(* IEC 61131-3 sources: simple-control-modules/test, 8 files *)

(* ---- AbstractEncoderTest.st ---- *)
USING AxUnit.Assert;
USING Simatic.Ax.SimpleControlModules;

NAMESPACE Simatic.Ax.SimpleControlModules
    CLASS EncoderTest EXTENDS Simatic.Ax.SimpleControlModules.AbstractEncoder
        VAR

        END_VAR

        METHOD PUBLIC OVERRIDE Evaluate
            ;
        END_METHOD
    END_CLASS
END_NAMESPACE

NAMESPACE Simatic.Ax.SimpleControlModules.Test
    {TestFixture}
    CLASS Test_AbstractEncoder

        VAR
            enc : EncoderTest;
        END_VAR

        {Test}
        METHOD PUBLIC SetValue_to_555_expect_GetValue_555

            enc.SetValue(LINT#555);

            Equal(expected := LINT#555, actual := enc.GetValue());
            Equal(expected := LINT#0, actual := enc.RelativeCount());
            enc.Reset();

            Equal(expected := LINT#0, actual := enc.GetValue());
            Equal(expected := LINT#0, actual := enc.RelativeCount());
        END_METHOD

        {Test}
        METHOD PUBLIC Test_Reset_Expect_value_0

            enc.SetValue(LINT#555);
            enc.Reset();

            Equal(expected := LINT#0, actual := enc.GetValue());
            Equal(expected := LINT#0, actual := enc.RelativeCount());
        END_METHOD

    END_CLASS

END_NAMESPACE

(* ---- CounterTest.st ---- *)
USING AxUnit.Assert;
USING AxUnit.Assert;
USING Simatic.Ax.SimpleControlModules;
NAMESPACE Simatic.Ax.SimpleControlModules.Test
    {TestFixture}
    CLASS TestCounterClass
        VAR
            cnt : Counter;
            cntStateLess : Counter;
        END_VAR

        {TestSetup}
        METHOD PUBLIC MyTestSetup
            // Will be called before MyTest_A AND before Test_B are executed
            cnt := cntStateLess;
        END_METHOD

        {Test}
        METHOD PUBLIC Count_Forward_3_times_Expect_3;
            cnt.CountForward();
            Equal(expected := 1, actual := cnt.CounterValue());
            cnt.CountForward();
            cnt.CountForward();
            Equal(expected := 3, actual := cnt.CounterValue());
        END_METHOD

        {Test}
        METHOD PUBLIC Count_Reverse_3_times_From_3_Expect_0;
            cnt.SetCounterValue(value := 3);
            Equal(expected := 3, actual := cnt.CounterValue());
            cnt.CountReverse();
            Equal(expected := 2, actual := cnt.CounterValue());
            cnt.CountReverse();
            cnt.CountReverse();
            Equal(expected := 0, actual := cnt.CounterValue());
        END_METHOD

        {Test}
        METHOD PUBLIC Count_Forward_3_times_by_2_Expect_3;
            cnt.CountForward(increment := 2);
            Equal(expected := 2, actual := cnt.CounterValue());
            cnt.CountForward(increment := 2);
            cnt.CountForward(increment := 2);
            Equal(expected := 6, actual := cnt.CounterValue());
        END_METHOD

        {Test}
        METHOD PUBLIC Count_Reverse_3_timesby_2_From_6_Expect_0;
            cnt.SetCounterValue(value := 6);
            Equal(expected := 6, actual := cnt.CounterValue());
            cnt.CountReverse(decrement := 2);
            Equal(expected := 4, actual := cnt.CounterValue());
            cnt.CountReverse(decrement := 2);
            cnt.CountReverse(decrement := 2);
            Equal(expected := 0, actual := cnt.CounterValue());
        END_METHOD

        {Test}
        METHOD PUBLIC Counter_Lower_Limit_Reached
            cnt.Config(ll := DINT#-4, ul := DINT#4);
            Equal(expected := FALSE, actual := cnt.LowerLimitReached());
            Equal(expected := FALSE, actual := cnt.UpperLimitReached());
            cnt.CountReverse();
            cnt.CountReverse();
            cnt.CountReverse();
            Equal(expected := FALSE, actual := cnt.LowerLimitReached());
            cnt.CountReverse();
            Equal(expected := TRUE, actual := cnt.LowerLimitReached());
            Equal(expected := FALSE, actual := cnt.UpperLimitReached());
        END_METHOD

        {Test}
        METHOD PUBLIC Counter_Lower_Limit_Reached_When_Limit_Is_1
            cnt.Config(ll := DINT#1, ul := DINT#4);
            Equal(expected := TRUE, actual := cnt.LowerLimitReached());
            Equal(expected := FALSE, actual := cnt.UpperLimitReached());
            cnt.CountReverse();
            cnt.CountReverse();
            cnt.CountReverse();
            Equal(expected := TRUE, actual := cnt.LowerLimitReached());
            cnt.CountReverse();
            Equal(expected := TRUE, actual := cnt.LowerLimitReached());
            Equal(expected := FALSE, actual := cnt.UpperLimitReached());
        END_METHOD

        {Test}
        METHOD PUBLIC Counter_Upper_Limit_Reached_When_UpperLimit_Is4
            cnt.Config(ll := DINT#-4, ul := DINT#4);
            Equal(expected := FALSE, actual := cnt.LowerLimitReached());
            Equal(expected := FALSE, actual := cnt.UpperLimitReached());
            cnt.CountForward();
            cnt.CountForward();
            cnt.CountForward();
            Equal(expected := FALSE, actual := cnt.UpperLimitReached());
            cnt.CountForward();
            Equal(expected := TRUE, actual := cnt.UpperLimitReached());
            Equal(expected := FALSE, actual := cnt.LowerLimitReached());
            cnt.CountReverse();
            Equal(expected := FALSE, actual := cnt.UpperLimitReached());
        END_METHOD

        {Test}
        METHOD PUBLIC Counter_Upper_Limit_Reached_When_UpperLimit_Is0
            cnt.Config(ll := DINT#-4, ul := DINT#0);
            Equal(expected := FALSE, actual := cnt.LowerLimitReached());
            Equal(expected := TRUE, actual := cnt.UpperLimitReached());
            cnt.CountForward();
            cnt.CountForward();
            cnt.CountForward();
            Equal(expected := TRUE, actual := cnt.UpperLimitReached());
            cnt.CountForward();
            Equal(expected := TRUE, actual := cnt.UpperLimitReached());
            Equal(expected := FALSE, actual := cnt.LowerLimitReached());
        END_METHOD
    END_CLASS
END_NAMESPACE

(* ---- EncoderABTest.st ---- *)
USING Simatic.Ax.IO.Input;
USING AxUnit.Assert;
USING Simatic.Ax.SimpleControlModules;
NAMESPACE Simatic.Ax.SimpleControlModules.Test
    {TestFixture}
    CLASS Test_EncoderAB IMPLEMENTS AxUnit.Mocking.IPayload

        VAR
            enc : EncoderAB;
            sigA : BinSignal;
            sigB : BinSignal;
            //signalMock : BinSignalQMockAB;

            signalsA : ARRAY[0..13] OF BOOL := [FALSE, TRUE, TRUE, FALSE, FALSE, TRUE, TRUE, FALSE, FALSE, TRUE, TRUE, FALSE, FALSE, TRUE];
            signalsB : ARRAY[0..13] OF BOOL := [FALSE, FALSE, TRUE, TRUE, FALSE, FALSE, TRUE, TRUE, FALSE, FALSE, TRUE, TRUE, FALSE, FALSE];

        END_VAR

        {Test}
        // Encoder Forward Test
        METHOD PUBLIC AB_Encoder_A_Forward_test_Expect_13
                VAR_TEMP
                    i : INT;
                END_VAR

                enc.SignalA := sigA;
                enc.SignalB := sigB;

                FOR i := 0 TO 13 DO
                    sigA.ReadCyclic(signal := signalsA[i]);
                    sigB.ReadCyclic(signal := signalsB[i]);
                    enc.Evaluate();
                END_FOR;

                Equal(expected := LINT#13, actual := enc.GetValue());
                Equal(expected := LINT#13, actual := enc.RelativeCount());
                ;
        END_METHOD

        // Encoder Count Reverse Test
        {Test}
        METHOD PUBLIC AB_Encoder_A_Reverse_test_Expect_Minus_13
            VAR_TEMP
                i : INT;
            END_VAR

            enc.SignalA := sigA;
            enc.SignalB := sigB;
            enc.SetDirection(mode := CountMode#Reverse);
            FOR i := 0 TO 13 DO
                sigA.ReadCyclic(signal := signalsA[i]);
                sigB.ReadCyclic(signal := signalsB[i]);

                enc.Evaluate();
            END_FOR;

            Equal(expected := LINT#-13, actual := enc.GetValue());
            Equal(expected := LINT#-13, actual := enc.RelativeCount());
            ;
        END_METHOD

        {Test}
        // Encoder Swap singnals Test
        METHOD PUBLIC AB_Encoder_Swap_AB_Signal_And_Expect_Minus_13
                VAR_TEMP
                    i : INT;
                END_VAR

                // Swap AB
                enc.SignalA := sigB;
                enc.SignalB := sigA;
                FOR i := 0 TO 13 DO
                    sigA.ReadCyclic(signal := signalsA[i]);
                    sigB.ReadCyclic(signal := signalsB[i]);
                    enc.Evaluate();
                END_FOR;

                Equal(expected := LINT#-13, actual := enc.GetValue());
                Equal(expected := LINT#-13, actual := enc.RelativeCount());
                ;
        END_METHOD

        // Encoder change signal sequence to reverse
        {Test}
        METHOD PUBLIC AB_Encoder_9_Forward_5_Reverse_expect
            VAR_TEMP
                i : INT;
            END_VAR

            enc.SignalA := sigA;
            enc.SignalB := sigB;

            FOR i := 0 TO 9 DO
                sigA.ReadCyclic(signal := signalsA[i]);
                sigB.ReadCyclic(signal := signalsB[i]);
                enc.Evaluate();
            END_FOR;

            Equal(expected := LINT#9, actual := enc.GetValue());

            FOR i := 9 TO 0 BY -1 DO
                sigA.ReadCyclic(signal := signalsA[i]);
                sigB.ReadCyclic(signal := signalsB[i]);
                enc.Evaluate();
            END_FOR;
            Equal(expected := LINT#0, actual := enc.GetValue());
            Equal(expected := LINT#0, actual := enc.RelativeCount());
            ;
        END_METHOD

        // Encoder Reverse Test
        {Test}
        METHOD PUBLIC AB_Encoder_9_Forward_4_Reverse_expet_5
            VAR_TEMP
                i : INT;
            END_VAR

            enc.SignalA := sigA;
            enc.SignalB := sigB;

            FOR i := 0 TO 9 DO
                sigA.ReadCyclic(signal := signalsA[i]);
                sigB.ReadCyclic(signal := signalsB[i]);

                enc.Evaluate();
            END_FOR;
            Equal(expected := LINT#9, actual := enc.GetValue());

            enc.SetDirection(mode := CountMode#Reverse);
            FOR i := 10 TO 13 DO
                sigA.ReadCyclic(signal := signalsA[i]);
                sigB.ReadCyclic(signal := signalsB[i]);
            enc.Evaluate();
            END_FOR;
            Equal(expected := LINT#5, actual := enc.GetValue());
            Equal(expected := LINT#5, actual := enc.RelativeCount());
            ;
        END_METHOD

        {Test}
        METHOD PUBLIC Single_Track_Test_Reset
            VAR_TEMP
                i : INT;
            END_VAR

            THIS.AB_Encoder_A_Forward_test_Expect_13();

            enc.Reset();
            Equal(expected := LINT#0, actual := enc.GetValue());
        END_METHOD

        {Test}
        METHOD PUBLIC AB_Encoder_RelativeValue
            VAR_TEMP
                i : INT;
            END_VAR

            // 3 Rising edges 3 Falling edges --> 6 pulses
            enc.SignalA := sigA;
            enc.SignalB := sigB;

            FOR i := 0 TO 9 DO
                sigA.ReadCyclic(signal := signalsA[i]);
                sigB.ReadCyclic(signal := signalsB[i]);
            enc.Evaluate();
            END_FOR;
            Equal(expected := LINT#9, actual := enc.GetValue());
            Equal(expected := LINT#9, actual := enc.RelativeCount());
            enc.ResetRelative();

            FOR i := 10 TO 13 DO
                sigA.ReadCyclic(signal := signalsA[i]);
                sigB.ReadCyclic(signal := signalsB[i]);
            enc.Evaluate();
            END_FOR;
            Equal(expected := LINT#13, actual := enc.GetValue());
            Equal(expected := LINT#4, actual := enc.RelativeCount());
            ;
        END_METHOD

    END_CLASS

END_NAMESPACE

(* ---- EncoderATest.st ---- *)
USING Simatic.Ax.IO.Input;
USING AxUnit.Assert;
USING Simatic.Ax.SimpleControlModules;

NAMESPACE Simatic.Ax.SimpleControlModules.Test
    {TestFixture}
    CLASS Test_EncoderA IMPLEMENTS AxUnit.Mocking.IPayload

        VAR
            enc : EncoderA;
            sig : BinSignal;
            signalMock : BinSignalQMock;
        END_VAR

        {Test}
        // Encoder Forward Test
        METHOD PUBLIC Single_Track_Encoder_A_Forward_test_Expect_6
                VAR_TEMP
                    i : INT;
                END_VAR

                // 3 Rising edges 3 Falling edges --> 6 pulses
                enc.SignalA := sig;
                FOR i := 0 TO 13 DO
                    sig.ReadCyclic(signal := signalMock.Q());
                    enc.Evaluate();
                END_FOR;

                Equal(expected := LINT#6, actual := enc.GetValue());
                Equal(expected := LINT#6, actual := enc.RelativeCount());
                ;
        END_METHOD

        // Encoder Reverse Test
        {Test}
        METHOD PUBLIC Single_Track_Encoder_A_Reverse_test_Expect_Minus_6
            VAR_TEMP
                i : INT;
            END_VAR

            // 3 Rising edges 3 Falling edges --> 6 pulses
            enc.SignalA := sig;
            enc.SetDirection(mode := CountMode#Reverse);
            FOR i := 0 TO 13 DO
                sig.ReadCyclic(signal := signalMock.Q());
                enc.Evaluate();
            END_FOR;

            Equal(expected := LINT#-6, actual := enc.GetValue());
            Equal(expected := LINT#-6, actual := enc.RelativeCount());
            ;
        END_METHOD

        // Encoder Reverse Test
        {Test}
        METHOD PUBLIC Single_Track_Encoder_4_Forward_2_Reverse_expet_2
            VAR_TEMP
                i : INT;
            END_VAR

            // 3 Rising edges 3 Falling edges --> 6 pulses
            enc.SignalA := sig;
            FOR i := 0 TO 9 DO
                sig.ReadCyclic(signal := signalMock.Q());
                enc.Evaluate();
            END_FOR;
            Equal(expected := LINT#4, actual := enc.GetValue());

            enc.SetDirection(mode := CountMode#Reverse);
            FOR i := 0 TO 3 DO
                sig.ReadCyclic(signal := signalMock.Q());
                enc.Evaluate();
            END_FOR;
            Equal(expected := LINT#2, actual := enc.GetValue());
            Equal(expected := LINT#2, actual := enc.RelativeCount());
            ;
        END_METHOD

        {Test}
        METHOD PUBLIC Single_Track_Test_Reset
            VAR_TEMP
                i : INT;
            END_VAR

            THIS.Single_Track_Encoder_A_Forward_test_Expect_6();

            enc.Reset();
            Equal(expected := LINT#0, actual := enc.GetValue());
        END_METHOD

        {Test}
        METHOD PUBLIC Single_Track_Encoder_RelativeValue
            VAR_TEMP
                i : INT;
            END_VAR

            // 3 Rising edges 3 Falling edges --> 6 pulses
            enc.SignalA := sig;
            FOR i := 0 TO 9 DO
                sig.ReadCyclic(signal := signalMock.Q());
                enc.Evaluate();
            END_FOR;
            Equal(expected := LINT#4, actual := enc.GetValue());
            Equal(expected := LINT#4, actual := enc.RelativeCount());
            enc.ResetRelative();

            FOR i := 0 TO 3 DO
                sig.ReadCyclic(signal := signalMock.Q());
                enc.Evaluate();
            END_FOR;
            Equal(expected := LINT#6, actual := enc.GetValue());
            Equal(expected := LINT#2, actual := enc.RelativeCount());
            ;
        END_METHOD

    END_CLASS

    CLASS BinSignalQMock
        VAR PUBLIC
            signal : BOOL;
            pos : INT;
            signals : ARRAY[0..13] OF BOOL := [FALSE, FALSE, TRUE, TRUE, FALSE, FALSE, TRUE, TRUE, FALSE, FALSE, TRUE, TRUE, FALSE, FALSE];
        END_VAR
        METHOD PUBLIC Q : BOOL
            Q := signals[pos];
            pos := pos + 1;
            pos := pos MOD 12;
            ;
        END_METHOD
    END_CLASS

END_NAMESPACE

(* ---- PusherBiDirTimebasedTest .st ---- *)
USING Simatic.Ax.IO.Output;
USING Simatic.Ax.IO.Output;
USING AxUnit.Assert;
USING Simatic.Ax.SimpleControlModules;

NAMESPACE Simatic.Ax.SimpleControlModules.Test
    {TestFixture}
    CLASS Test_PusherBiDirTimeBased // IMPLEMENTS AxUnit.Mocking.IPayload

        VAR
            pusher : PusherBiDirTimeBased := (OnDuration := T#5s, OffDuration := T#5s);
            sig : BinOutput;
            sigOff : BinOutput;
            q : BOOL;
        END_VAR

        METHOD PUBLIC Setup
            pusher.ControlPush := sig;
            pusher.ControlRetract := sigOff;
        END_METHOD

        {Test}
        // Initial State
        METHOD PUBLIC Initial_State_expect_Retracted
            THIS.Setup();
            Equal(expected := TRUE, actual :=  pusher.GetState() = PusherState#Retracted);
            Equal(expected := FALSE, actual :=  q);
            pusher.Evaluate();
            Equal(expected := TRUE, actual :=  pusher.GetState() = PusherState#Retracted);
            Equal(expected := FALSE, actual :=  sig.IsOn());
        END_METHOD

        {Test}
        // Test Pushing
        METHOD PUBLIC Push_Expect_State_Pushing_Q_TRUE
            THIS.Setup();
            pusher.Push();
            pusher.Evaluate();
            Equal(expected := TRUE, actual :=  pusher.GetState() = PusherState#Pushing);
            Equal(expected := TRUE, actual :=  sig.IsOn());
        END_METHOD

        // {Test}
        // METHOD PUBLIC Retract_After_time
        //     THIS.Push_Expect_State_Pushing_Q_TRUE();
        //     AxUnit.Mocking.Mock(name_of(System.Timer.OnDelay), name_of(Simatic.Ax.Mocks.OnDelayMock_true));
        //     pusher.Evaluate();
        //     Equal(expected := TRUE, actual :=  pusher.GetState() = PusherState#Pushed);
        //     Equal(expected := TRUE, actual :=  sig.IsOn());
        //     Equal(expected := FALSE, actual :=  sigOff.IsOn());
        //     pusher.Evaluate();
        //     // Equal(expected := TRUE, actual :=  pusher.GetState() = PusherState#Retracting);
        //     // Equal(expected := FALSE, actual :=  sig.IsOn());
        //     // Equal(expected := TRUE, actual :=  sigOff.IsOn());
        //     // pusher.Evaluate();
        //     // Equal(expected := TRUE, actual :=  pusher.GetState() = PusherState#Retracted);
        //     // Equal(expected := FALSE, actual :=  sig.IsOn());
        //     // Equal(expected := FALSE, actual :=  sigOff.IsOn());
        // END_METHOD

    END_CLASS

END_NAMESPACE

(* ---- PusherTimebasedTest.st ---- *)
USING Simatic.Ax.IO.Output;
USING Simatic.Ax.IO.Output;
USING AxUnit.Assert;
USING Simatic.Ax.SimpleControlModules;

NAMESPACE Simatic.Ax.SimpleControlModules.Test
    {TestFixture}
    CLASS Test_PusherTimeBased // IMPLEMENTS AxUnit.Mocking.IPayload

        VAR
            pusher : PusherTimeBased := (OnDuration := T#5s);
            sig : BinOutput;
            q : BOOL;
        END_VAR

        METHOD PUBLIC Setup
            pusher.ControlPush := sig;
        END_METHOD

        {Test}
        // Initial State
        METHOD PUBLIC Initial_State_expect_Retracted
            THIS.Setup();
            Equal(expected := TRUE, actual :=  pusher.GetState() = PusherState#Retracted);
            Equal(expected := FALSE, actual :=  q);
            pusher.Evaluate();
            Equal(expected := TRUE, actual :=  pusher.GetState() = PusherState#Retracted);
            Equal(expected := FALSE, actual :=  sig.IsOn());
        END_METHOD

        {Test}
        // Test Pushing
        METHOD PUBLIC Push_Expect_State_Pushing_Q_TRUE
            THIS.Setup();
            pusher.Push();
            pusher.Evaluate();
            Equal(expected := TRUE, actual :=  pusher.GetState() = PusherState#Pushing);
            Equal(expected := TRUE, actual :=  sig.IsOn());
        END_METHOD

        // {Test}
        // METHOD PUBLIC Retract_After_time
        //     THIS.Push_Expect_State_Pushing_Q_TRUE();
        //     AxUnit.Mocking.Mock(name_of(System.Timer.OnDelay), name_of(Simatic.Ax.Mocks.OnDelayMock_true));
        //     pusher.Evaluate();
        //     Equal(expected := TRUE, actual :=  pusher.GetState() = PusherState#Retracting);
        //     Equal(expected := FALSE, actual :=  sig.IsOn());
        //     pusher.Evaluate();
        //     Equal(expected := TRUE, actual :=  pusher.GetState() = PusherState#Retracted);
        // END_METHOD

    END_CLASS

END_NAMESPACE

(* ---- TestBulb.st ---- *)
USING AxUnit.Assert;
USING Simatic.Ax.Io.Output;
USING Simatic.Ax.Io;
USING AxUnit.Assert;

NAMESPACE Simatic.Ax.SimpleControlModules.Test
    {TestFixture}
    CLASS TestClassBulb
        VAR PRIVATE
            b : Bulb;
            o : BinOutput;
            q : BOOL;
        END_VAR

        {Test}
        METHOD PUBLIC TestSwitchOn
            b.Output := o;
            Equal(expected := FALSE, actual := q);
            b.SwitchOn();
            o.WriteCyclic(q);
            Equal(expected := TRUE, actual := q);
        END_METHOD

        {Test}
        METHOD PUBLIC TestSwitchOff
            this.TestSwitchOn();

            Equal(expected := TRUE, actual := q);
            b.SwitchOff();
            o.WriteCyclic(q);
            Equal(expected := FALSE, actual := q);
        END_METHOD

        {Test}
        METHOD PUBLIC TestSwitchToggle
            this.TestSwitchOn();

            Equal(expected := TRUE, actual := q);
            b.Toggle();
            o.WriteCyclic(q);
            Equal(expected := FALSE, actual := q);
            b.Toggle();
            o.WriteCyclic(q);
            Equal(expected := TRUE, actual := q);
        END_METHOD

    END_CLASS
END_NAMESPACE

(* ---- TestLightStackRdYeGn.st ---- *)
USING AxUnit.Assert;
USING Simatic.Ax.Io.Output;
USING Simatic.Ax.Io;
USING AxUnit.Assert;

NAMESPACE Simatic.Ax.SimpleControlModules.Test
    {TestFixture}
    CLASS TestLightStackRdYeGnBl
        VAR PRIVATE
            o : LightStackRdYeGnBl;
            QRed : BinOutput;
            QYellow : BinOutput;
            QGreen : BinOutput;
            QBlue : BinOutput;
        END_VAR

        METHOD PRIVATE Init
            o.QRed := QRed;
            o.QYellow := QYellow;
            o.QGreen := QGreen;
            o.QBlue := QBlue;
        END_METHOD

        {Test}
        METHOD PUBLIC InitialState
            THIS.Init();
            Equal(expected := FALSE, actual := o.GetState(Colors#Red));
            Equal(expected := FALSE, actual := o.GetState(Colors#Yellow));
            Equal(expected := FALSE, actual := o.GetState(Colors#Green));
            Equal(expected := FALSE, actual := o.GetState(Colors#Blue));
        END_METHOD
        {Test}
        METHOD PUBLIC TestSwitchOnRed_Expect_True
            THIS.Init();
            Equal(expected := FALSE, actual := o.GetState(Colors#Red));
            o.SwitchOn(Colors#Red);
            Equal(expected := TRUE, actual := o.GetState(Colors#Red));
            Equal(expected := FALSE, actual := o.GetState(Colors#Yellow));
            Equal(expected := FALSE, actual := o.GetState(Colors#Green));
            Equal(expected := FALSE, actual := o.GetState(Colors#Blue));
            o.SwitchOff(Colors#Red);
            Equal(expected := FALSE, actual := o.GetState(Colors#Red));
        END_METHOD
        {Test}
        METHOD PUBLIC TestSwitchOnyellowExpect_True
            THIS.Init();
            Equal(expected := FALSE, actual := o.GetState(Colors#Yellow));
            o.SwitchOn(Colors#Yellow);
            Equal(expected := FALSE, actual := o.GetState(Colors#Red));
            Equal(expected := TRUE, actual := o.GetState(Colors#Yellow));
            Equal(expected := FALSE, actual := o.GetState(Colors#Green));
            Equal(expected := FALSE, actual := o.GetState(Colors#Blue));
            o.SwitchOff(Colors#Yellow);
            Equal(expected := FALSE, actual := o.GetState(Colors#Yellow));
        END_METHOD
        {Test}
        METHOD PUBLIC TestSwitchOnGreenExpect_True
            THIS.Init();
            Equal(expected := FALSE, actual := o.GetState(Colors#Green));
            o.SwitchOn(Colors#Green);
            Equal(expected := FALSE, actual := o.GetState(Colors#Red));
            Equal(expected := FALSE, actual := o.GetState(Colors#Yellow));
            Equal(expected := TRUE, actual := o.GetState(Colors#Green));
            Equal(expected := FALSE, actual := o.GetState(Colors#Blue));
            o.SwitchOff(Colors#Green);
            Equal(expected := FALSE, actual := o.GetState(Colors#Green));
        END_METHOD
        {Test}
        METHOD PUBLIC TestSwitchOnBlueExpect_True
            THIS.Init();
            Equal(expected := FALSE, actual := o.GetState(Colors#Blue));
            o.SwitchOn(Colors#Blue);
            Equal(expected := FALSE, actual := o.GetState(Colors#Red));
            Equal(expected := FALSE, actual := o.GetState(Colors#Yellow));
            Equal(expected := FALSE, actual := o.GetState(Colors#Green));
            Equal(expected := TRUE, actual := o.GetState(Colors#Blue));
            o.SwitchOff(Colors#Blue);
            Equal(expected := FALSE, actual := o.GetState(Colors#Blue));
        END_METHOD
    END_CLASS
END_NAMESPACE
